FUNCTION_BLOCK Forces5
VAR_INPUT
END_VAR
VAR_OUTPUT
END_VAR
VAR
END_VAR

END_FUNCTION_BLOCK

(* stored: Version 1.1.0.1, ProductVersion 3.1.4024.11
   POU Forces5: Id {4acd2301-6cae-4c87-b50e-09f23b809773}, SpecialFunc None *)
